FUNCTION TryConvert_TIME_TO_LWORD : BOOL
VAR_INPUT
	in : TIME;
	out : REFERENCE TO LWORD;
END_VAR

out := TIME_TO_LWORD(in);
TryConvert_TIME_TO_LWORD := TRUE;

END_FUNCTION

(* stored: Version 1.1.0.1, ProductVersion 3.1.4024.12
   POU TryConvert_TIME_TO_LWORD: Id {ead96845-b2b4-4b3c-a241-0217581871af}, SpecialFunc None *)
